//{attribute 'qualified_only'}
VAR_GLOBAL
	uIOLINK1 AT%Q* : ULINT;
	uIOLINK2 AT%Q* : ULINT;	

	inputs AT %I* : ARRAY [1..4] OF EL1809;
	outputs AT %Q* : ARRAY[1..1] OF EL2809;
	
	//manifold AT %Q* : ARRAY[1..3] OF ST_VTUG;

END_VAR

(* stored: Version 1.1.0.1, ProductVersion 3.1.4024.12
   GVL GVL_IO: Id {8dfeac7d-881a-4ac7-9fd5-d9954263b863} *)
